(* CODESYS project 06_MySQL_DB_Internal.ecp

Project tree, tasks and I/O mapping:
  PFC200_CS_2ETH_RS : 750-8212 PFC200 G2 2ETH RS, WAGO, order no. 0750-8212, version 5.16.3.16
    application Application
      libraries: ; WagoAppTime, 1.7.3.3 (WAGO); WagoAppSQL_MySQL, 1.6.1.0 (WAGO); SysProcess, 3.5.16.0 (System)
      task Task_SQL (cyclic, interval t#100ms, priority 14) calls PRG_SQL
      program PRG_SQL [FBD]
      Funktionen/
        function FuBuildSQLCommand_Concat [ST]
        function FuBuildSQLCommand_Concat9 [ST]
      Funktionsbausteine/
        function block FbSQLInsertCommand [ST]
      other/
        function FuBuildSQLCommand_Format9 [ST]
    ProjectConfiguration
    ProjectConfigurationTxt
    Kbus : Kbus, WAGO, version 1.4.0.2
        unmapped channels: K-BUS diagnostics
    MODBUS
      MODBUS : MODBUS, WAGO, order no. n/a, version 1.1.1.16
    Serial
      COM1 : COM1, WAGO, version 0.0.0.19
    Common.PCI
    EtherNet/IP
      Ethernet : Ethernet, WAGO, version 35.16.0.0
  00000000-0000-0000-0000-000000000000|C:\Users\MarkusF\AppData\Local\Temp\055e7d9746fd4311b0b4a460269c1d9c\Project.xml
  00000000-0000-0000-0000-000000000000|C:\Users\MarkusF\AppData\Local\Temp\1759141298bb48ef90c244c8cfde3aed\ProjectCfg.txt
*)

// PFC200_CS_2ETH_RS/Application/PRG_SQL
PROGRAM PRG_SQL
VAR
//_______________________________________________________________

	oFbInternalSQL		: FbSQLInsertCommand;
	sInternalSQLDB		: STRING := '127.0.0.1';		// localhost
	xConnect01			: BOOL;							// stays true
	sUsername			: STRING(30) := 'admin';
	sPassword			: STRING(30) := 'wago';
	sDatabase			: STRING(30) := 'dbInternal';
	sTable				: STRING(30) := 'dbPFC_Data';
	xTriggerWrite01		: BOOL;							// will get true and on completion be reset
	sStatus_dbInternal	: STRING;
//_______________________________________________________________
END_VAR

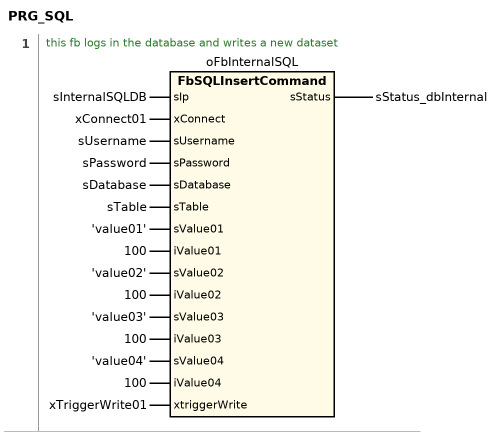
// NETWORK 1
// this fb logs in the database and writes a new dataset
oFbInternalSQL(
    sIp := sInternalSQLDB,
    xConnect := xConnect01,
    sUsername := sUsername,
    sPassword := sPassword,
    sDatabase := sDatabase,
    sTable := sTable,
    sValue01 := 'value01',
    iValue01 := 100,
    sValue02 := 'value02',
    iValue02 := 100,
    sValue03 := 'value03',
    iValue03 := 100,
    sValue04 := 'value04',
    iValue04 := 100,
    xtriggerWrite := xTriggerWrite01); // FbSQLInsertCommand
sStatus_dbInternal := oFbInternalSQL.sStatus;

END_PROGRAM

// PFC200_CS_2ETH_RS/Application/Funktionsbausteine/FbSQLInsertCommand
FUNCTION_BLOCK FbSQLInsertCommand
VAR_INPUT
	sIp:			STRING := '127.0.0.1';
	xConnect:		BOOL;
	sUsername:		STRING;
	sPassword:		STRING;
	sDatabase:		STRING;
	sTable:			STRING;
	
	sValue01:		STRING;		// first column
	iValue01:		INT;
	
	sValue02:		STRING;		// second column
	iValue02:		INT;
	
	sValue03:		STRING;		// third column
	iValue03:		INT;
	
	sValue04:		STRING;		// fourth column
	iValue04:		INT;
END_VAR
VAR_OUTPUT
	sStatus:		STRING;
END_VAR
VAR_IN_OUT
	xtriggerWrite:	BOOL;
END_VAR
VAR
	R1				: R_TRIG;
	F1				: F_TRIG;
	index			: INT;	// used by the state machine to determine the current state

	mySqlString_Format9: MaxString;
	
	Login01			: FbMySql_Login;
	xTriggerLogin	: BOOL;	
	xBusyLogIn		: BOOL;	
	xErrorLogIn		: BOOL;
	sStatusLogIn	: STRING(200);
	xConnected		: BOOL;

	Exec01			: FbMySql_Execute;
	aSqlCommand		: ARRAY [0..MYSQL_SQL_UPPER_BOUND] OF STRING(MYSQL_SQL_LENGTH);
	mySqlString		: STRING(255);
	mySqlString_Concat9: MaxString;
	xBusyWrite		: BOOL;
	xErrorWrite		: BOOL;
	sStatusWrite	: STRING(200);

	Logout01		: FbMySql_Logout;
	xTriggerLogout	: BOOL;	
	xBusyLogOut		: BOOL;
	xErrorLogOut	: BOOL;
	sStatusLogOut	: STRING(200);
END_VAR

R1(CLK := xConnect);
F1(CLK := xConnect);

// target string:  'INSERT INTO dbInternal(value01,value02,value03,value04) VALUES(100,200,300,400)';

(*
mySqlString := FuBuildSQLCommand_Concat(
	sTable	 := sTable,
	sValue01 := sValue01,
	iValue01 := iValue01 + 1,
	sValue02 := sValue02,
	iValue02 := iValue02 + 1,
	sValue03 := sValue03,
	iValue03 := iValue03 + 1,
	sValue04 := sValue04,
	iValue04 := iValue04 + 1);
*)

(*	
mySqlString := FuBuildSQLCommand_Concat9(
	sTable	 := sTable,
	sValue01 := sValue01,
	iValue01 := iValue01 + 2,
	sValue02 := sValue02,
	iValue02 := iValue02 + 2,
	sValue03 := sValue03,
	iValue03 := iValue03 + 2,
	sValue04 := sValue04,
	iValue04 := iValue04 + 2);
*)

mySqlString := FuBuildSQLCommand_Format9(
	sTable	:= sTable,
	sValue01:= sValue01,
	iValue01:= iValue01 + 3,
	sValue02:= sValue02,
	iValue02:= iValue02 + 3,
	sValue03:= sValue03,
	iValue03:= iValue03 + 3,
	sValue04:= sValue04,
	iValue04:= iValue04 + 3);

//-------state machine--------------//

IF R1.Q THEN
	index := 10;
END_IF

IF F1.Q THEN
	index := 100;
END_IF

CASE index OF
	0:
		sStatus := 'SQL_idle';
	
	10:
		xTriggerLogin := TRUE;
		index := 20;
	
	20:
		Login01(
			sHost		:= sIp,
			//uiPort	:=,
			sUsername	:= sUsername,
			sPassword	:= sPassword,
			sDatabase	:= sDatabase,
			xTrigger	:= xTriggerLogin,
			xBusy		=> xBusyLogIn,
			xError		=> xErrorLogIn,
			//oStatus	=> ,
			sStatus		=> sStatusLogIn,
			xConnected	=> xConnected);
		
		IF NOT xTriggerLogin THEN
			IF xConnected THEN
				index := 30;
				sStatus := 'SQL_connected';
			ELSE
				sStatus:='SQL_connect_error';
			index := 1000;
			END_IF
		END_IF
	
	30:
		aSqlCommand[0] := mySqlString;
		
		Exec01(
			aSqlCommand	:= aSqlCommand,
			xTrigger	:= xtriggerWrite,
			xBusy		=> xBusyWrite,
			xError		=> xErrorWrite,
			//oStatus	=> ,
			sStatus		=> sStatusWrite);
	
	100:
		xTriggerLogout := TRUE;
		index := 110;
	
	110:
		Logout01(
			xTrigger	:= xTriggerLogout,
			xBusy		=> xBusyLogOut,
			xError		=> xErrorLogOut,
			//oStatus	=> ,
			sStatus		=> sStatusLogOut);
		IF NOT xErrorLogOut THEN
			sStatus := 'SQL_disconnected';
			index := 0;
		ELSE
			sStatus := 'SQL_Logout_Error';
			index := 0;
		END_IF;
	
END_CASE

END_FUNCTION_BLOCK

// PFC200_CS_2ETH_RS/Application/Funktionen/FuBuildSQLCommand_Concat
FUNCTION FuBuildSQLCommand_Concat : STRING(255)		// not used here
VAR_INPUT
	sTable	: STRING(20);
	sValue01: STRING(20);
	iValue01: INT;
	sValue02: STRING(20);
	iValue02: INT;
	sValue03: STRING(20);
	iValue03: INT;
	sValue04: STRING(20);
	iValue04: INT;
END_VAR
VAR
	mySqlString: STRING(255);
END_VAR

mySqlString := CONCAT('INSERT INTO ', sTable); 							// INSERT INTO dbPFCData
mySqlString := CONCAT(mySqlString, '(');								// INSERT INTO dbPFCData(
mySqlString := CONCAT(CONCAT(mySqlString, sValue01), ',');				// INSERT INTO dbPFCData(value01
mySqlString := CONCAT(CONCAT(mySqlString, sValue02), ',');				// INSERT INTO dbPFCData(value01,value02
mySqlString := CONCAT(CONCAT(mySqlString, sValue03), ',');				// INSERT INTO dbPFCData(value01,value02,value03
mySqlString := CONCAT(CONCAT(mySqlString, sValue04), ')');				// INSERT INTO dbPFCData(value01,value02,value03,value04)

mySqlString := CONCAT(mySqlString, ' VALUES(');							// INSERT INTO dbPFCData(value01,value02,value03,value04) VALUES(
mySqlString := CONCAT(mySqlSTRING, 			   TO_STRING(iValue01));	// INSERT INTO dbPFCData(value01,value02,value03,value04) VALUES(1000
mySqlString := CONCAT(CONCAT(mySqlSTRING,','), TO_STRING(iValue02));	// INSERT INTO dbPFCData(value01,value02,value03,value04) VALUES(1000,2000
mySqlString := CONCAT(CONCAT(mySqlSTRING,','), TO_STRING(iValue03));	// INSERT INTO dbPFCData(value01,value02,value03,value04) VALUES(1000,2000,3000
mySqlString := CONCAT(CONCAT(mySqlSTRING,','), TO_STRING(iValue04));	// INSERT INTO dbPFCData(value01,value02,value03,value04) VALUES(1000,2000,3000,4000
mySqlString := CONCAT(mySqlString, ')');								// INSERT INTO dbPFCData(value01,value02,value03,value04) VALUES(1000,2000,3000,4000)

FuBuildSQLCommand_Concat := mySqlString;

END_FUNCTION

// PFC200_CS_2ETH_RS/Application/Funktionen/FuBuildSQLCommand_Concat9
FUNCTION FuBuildSQLCommand_Concat9 : STRING(255)		// not used here
VAR_INPUT
	sTable:   STRING(20);
	sValue01: STRING(20);
	iValue01: INT;
	sValue02: STRING(20);
	iValue02: INT;
	sValue03: STRING(20);
	iValue03: INT;
	sValue04: STRING(20);
	iValue04: INT;
END_VAR
VAR
	mySqlString_Concat9: STRING(255);
END_VAR

mySqlString_Concat9 := Concat9(
	s1 := 'INSERT INTO ',	// INSERT INTO 
	s2 := sTable, 			// INSERT INTO dbPFCData
	s3 := '(', 				// INSERT INTO dbPFCData(
	s4 := sValue01, 		// INSERT INTO dbPFCData(value01
	s5 := ',', 				// INSERT INTO dbPFCData(value01,	
	s6 := sValue02, 		// INSERT INTO dbPFCData(value01,value02
	s7 := ',', 				// INSERT INTO dbPFCData(value01,value02,
	s8 := sValue03, 		// INSERT INTO dbPFCData(value01,value02,value03
	s9 := ',');				// INSERT INTO dbPFCData(value01,value02,value03,

mySqlString_Concat9 := Concat9(
	s1 := mySqlString_Concat9,	// INSERT INTO dbPFCData(value01,value02,value03,
	s2 := sValue04, 			// INSERT INTO dbPFCData(value01,value02,value03,value04
	s3 := ') ', 				// INSERT INTO dbPFCData(value01,value02,value03,value04) 
	s4 := 'VALUES(', 			// INSERT INTO dbPFCData(value01,value02,value03,value04) VALUES(
	s5 := TO_STRING(iValue01), 	// INSERT INTO dbPFCData(value01,value02,value03,value04) VALUES(1000
	s6 := ',', 					// INSERT INTO dbPFCData(value01,value02,value03,value04) VALUES(1000,
	s7 := TO_STRING(iValue02), 	// INSERT INTO dbPFCData(value01,value02,value03,value04) VALUES(1000,2000
	s8 := ',', 					// INSERT INTO dbPFCData(value01,value02,value03,value04) VALUES(1000,2000,
	s9 := TO_STRING(iValue03), 	// INSERT INTO dbPFCData(value01,value02,value03,value04) VALUES(1000,2000,3000
	);

mySqlString_Concat9 := Concat4(
	s1 := mySqlString_Concat9,	// INSERT INTO dbPFCData(value01,value02,value03,value04) VALUES(1000,2000,3000
	s2 := ',',					// INSERT INTO dbPFCData(value01,value02,value03,value04) VALUES(1000,2000,3000,
	s3 := TO_STRING(iValue04), 	// INSERT INTO dbPFCData(value01,value02,value03,value04) VALUES(1000,2000,3000,4000
	s4 := ')', 					// INSERT INTO dbPFCData(value01,value02,value03,value04) VALUES(1000,2000,3000,4000)
	);

FuBuildSQLCommand_Concat9 := mySqlString_Concat9;

END_FUNCTION

// PFC200_CS_2ETH_RS/Application/other/FuBuildSQLCommand_Format9
FUNCTION FuBuildSQLCommand_Format9 : STRING(255)
VAR_INPUT
	sTable:   STRING(20);
	sValue01: STRING(20);
	iValue01: INT;
	sValue02: STRING(20);
	iValue02: INT;
	sValue03: STRING(20);
	iValue03: INT;
	sValue04: STRING(20);
	iValue04: INT;
END_VAR
VAR
	mySqlString_Format9: STRING(255);
END_VAR
(*
mySqlString_Format9:=Format9(
	
	sFormat:= 'INSERT INTO %s(%s,%s,%s,%s)VALUES(%i,%i,%i,%i)',	
    p1:= ADR(sTable), _____|  |  |  |   |         |  |  |  |
	p2:= ADR(sValue01),	______|  |  |	|		  |	 |	|  |						
	p3:= ADR(sValue02),__________|	|	|		  |	 |  |  | 			
	p4:= ADR(sValue03), ____________|   |         |  |  |  | 
	p5:= ADR(sValue04),_________________|		  |  |  |  |    
 												  |  |  |  |   
	p6:= ADR(iValue01),___________________________|  |  |  |    
	p7:= ADR(iValue02),______________________________|  |  | 
	p8:= ADR(iValue03),_________________________________|  |
	p9:= ADR(iValue04)_____________________________________|
);

    p1:= ADR(sTable),  //INSERT INTO dbPFCData(<sValue01>,<sValue02>,<sValue03>,<sValue04>)VALUES(<iValue01>,<iValue02>,<iValue03>,<iValue04>)
	p2:= ADR(sValue01),//INSERT INTO dbPFCData(value01   ,<sValue02>,<sValue03>,<sValue04>)VALUES(<iValue01>,<iValue02>,<iValue03>,<iValue04>) 															
	p3:= ADR(sValue02),//INSERT INTO dbPFCData(value01   ,value02   ,<sValue03>,<sValue04>)VALUES(<iValue01>,<iValue02>,<iValue03>,<iValue04>) 									
	p4:= ADR(sValue03),//INSERT INTO dbPFCData(value01   ,value02   ,value03   ,<sValue04>)VALUES(<iValue01>,<iValue02>,<iValue03>,<iValue04>) 
	p5:= ADR(sValue04),//INSERT INTO dbPFCData(value01   ,value02   ,value03   ,value04)   VALUES(<iValue01>,<iValue02>,<iValue03>,<iValue04>)
 
	p6:= ADR(iValue01),//INSERT INTO dbPFCData(value01   ,value02   ,value03   ,value04)   VALUES(1000     ,<iValue02>,<iValue03>,<iValue04>)
	p7:= ADR(iValue02),//INSERT INTO dbPFCData(value01   ,value02   ,value03   ,value04)   VALUES(1000     ,2000      ,<iValue03>,<iValue04>)
	p8:= ADR(iValue03),//INSERT INTO dbPFCData(value01   ,value02   ,value03   ,value04)   VALUES(1000     ,2000     ,3000      ,<iValue04>)
	p9:= ADR(iValue04)//INSERT INTO  dbPFCData(value01    ,value02   ,value03   ,value04)   VALUES(1000     ,2000     ,3000      ,4000)
);

*)

mySqlString_Format9:=Format9(
	
	sFormat := 'INSERT INTO %s(%s,%s,%s,%s)VALUES(%i,%i,%i,%i)',
	
    p1 := ADR(sTable),
	p2 := ADR(sValue01),
	p3 := ADR(sValue02),
	p4 := ADR(sValue03),
	p5 := ADR(sValue04),

	p6 := ADR(iValue01),
	p7 := ADR(iValue02),
	p8 := ADR(iValue03),
	p9 := ADR(iValue04));

FuBuildSQLCommand_Format9 := mySqlString_Format9;

END_FUNCTION
